TYPE McSetPositionProcessArgs :
STRUCT
	///New position to be taken over by the encoder
	value: LREAL;
END_STRUCT
END_TYPE

(* stored: Version 1.1.0.1, ProductVersion 3.1.4019.2
   DUT McSetPositionProcessArgs: Id {408b6075-cb63-4bd3-a784-0083170659f3} *)
